FUNCTION_BLOCK FB_REAL_UINT (* REAL to UINT conversion with limiting *)
  (* Standard: 61499-1 *)
  (* Version 0.1, 2001-04-21, JHC, Rockwell Automation, XML version. *)
  (* Version 0.0, 1999-01-10, JHC, Rockwell Automation, pre-XML version. *)
  (* Compiler header: package fb.rt.math; *)
  (* Compiler Java IBM VisualAge 3.0 *)
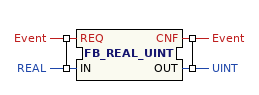
  EVENT_INPUT
    REQ WITH IN;
  END_EVENT
  EVENT_OUTPUT
    CNF WITH OUT;
  END_EVENT
  VAR_INPUT
    IN : REAL;
  END_VAR
  VAR_OUTPUT
    OUT : UINT;
  END_VAR
END_FUNCTION_BLOCK
